(* Logix 5000 project; controller cal1632 1756-L62 rev 16.20; software revision 16.05; part 49 of 57 *)
(* tags used below, declared in another part *)
   FAULT : BOOL;
   HMI : BOOL;
   p01_recipe_active : recipe;
   p01r09_pb_global_reset : BOOL;
   p01r09_request_line_jog : BOOL;
   p01r12_master_ramped_speed : REAL;
   p01r13_line_running : BOOL;
   p01r13_line_slow_ramp : BOOL;
   p01r13_permissive_drives : BOOL;
   p02_dint_from_hmi : hmi_dint;
   p25r11_request_thread_fwd : BOOL;
   p25r11_request_thread_rev : BOOL;
   p28_ai_slitter_amps : REAL;
   p28_ai_slitter_hz : REAL;
   p28_ai_slitter_speed : REAL;
   p28_ao_sltr_selected_speed : REAL;
   p28_di_brake : BOOL;
   p28_di_motor : BOOL;
   p28_di_slitter : acs800_di_normal;
   p28_dint_to_hmi : DINT[16];
   p28_do_sltr : acs800_do_normal;
   p28_real_to_hmi : REAL[112];
   p28_slitter_on : SYS_Toggle;
   p28r06 : routine;
   p28r06_timer_fault : TIMER[4];
   p28r06_timer_warning : TIMER[4];
   p28r07 : routine;
   p28r07_timer_fault : TIMER[4];
   p28r07_timer_warning : TIMER[4];
   p28r08 : routine;
   p28r08_timer_fault : TIMER[4];
   p28r08_timer_warning : TIMER[4];
   p28r09 : routine;
   p28r09_timer_fault : TIMER[4];
   p28r09_timer_warning : TIMER[4];
   p28r11 : routine;
   p28r11_permissive_run : BOOL;
   p28r11_request_line_jog : BOOL;
   p28r11_request_run : BOOL;
   p28r11_request_thread_fwd : BOOL;
   p28r11_request_thread_rev : BOOL;
   p28r11_slitter_on : BOOL;
   p28r11_timer_fault : TIMER[10];
   p28r11_timer_warning : TIMER[5];
(* P28_Slitter, continued *)

ROUTINE R06_Real_to_HMI   (* ladder *)
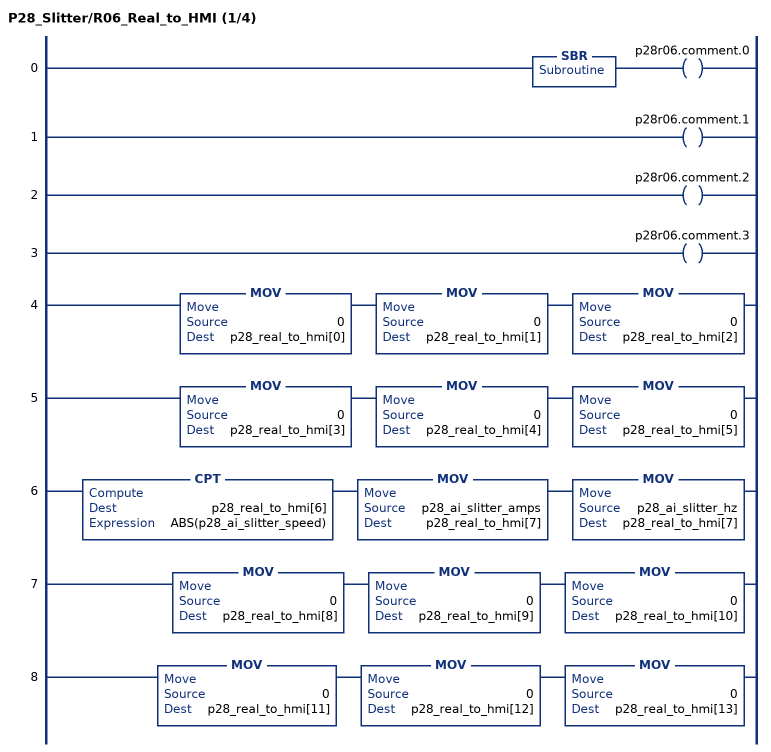
   0: SBR()OTE(p28r06.comment.0);
   1: OTE(p28r06.comment.1);
   2: OTE(p28r06.comment.2);
   3: OTE(p28r06.comment.3);
   4: MOV(0,p28_real_to_hmi[0])MOV(0,p28_real_to_hmi[1])MOV(0,p28_real_to_hmi[2]);
   5: MOV(0,p28_real_to_hmi[3])MOV(0,p28_real_to_hmi[4])MOV(0,p28_real_to_hmi[5]);
   6: CPT(p28_real_to_hmi[6],ABS(p28_ai_slitter_speed))MOV(p28_ai_slitter_amps,p28_real_to_hmi[7])MOV(p28_ai_slitter_hz,p28_real_to_hmi[7]);
   7: MOV(0,p28_real_to_hmi[8])MOV(0,p28_real_to_hmi[9])MOV(0,p28_real_to_hmi[10]);
   8: MOV(0,p28_real_to_hmi[11])MOV(0,p28_real_to_hmi[12])MOV(0,p28_real_to_hmi[13]);
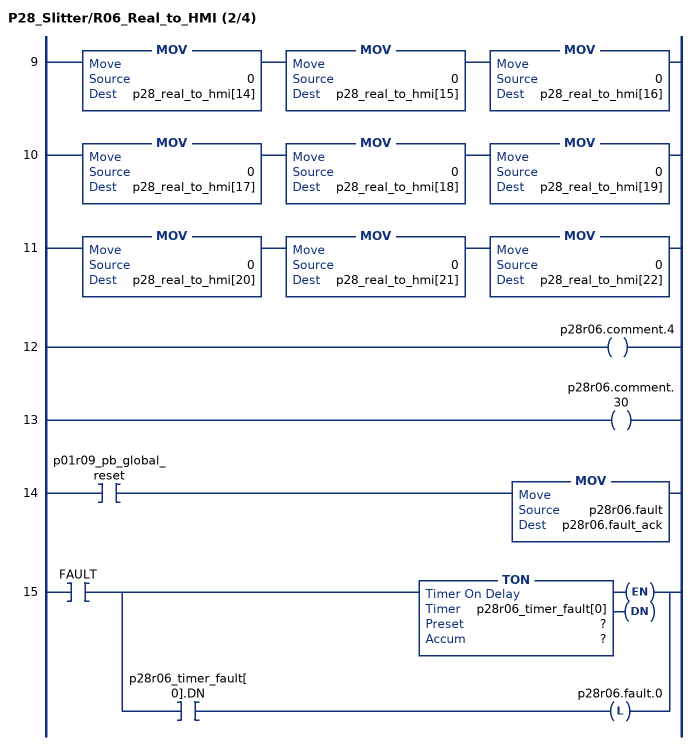
   9: MOV(0,p28_real_to_hmi[14])MOV(0,p28_real_to_hmi[15])MOV(0,p28_real_to_hmi[16]);
   10: MOV(0,p28_real_to_hmi[17])MOV(0,p28_real_to_hmi[18])MOV(0,p28_real_to_hmi[19]);
   11: MOV(0,p28_real_to_hmi[20])MOV(0,p28_real_to_hmi[21])MOV(0,p28_real_to_hmi[22]);
   12: OTE(p28r06.comment.4);
   13: OTE(p28r06.comment.30);
   14: XIC(p01r09_pb_global_reset)MOV(p28r06.fault,p28r06.fault_ack);
   15: XIC(FAULT)[TON(p28r06_timer_fault[0],?,?) ,XIC(p28r06_timer_fault[0].DN) OTL(p28r06.fault.0) ];
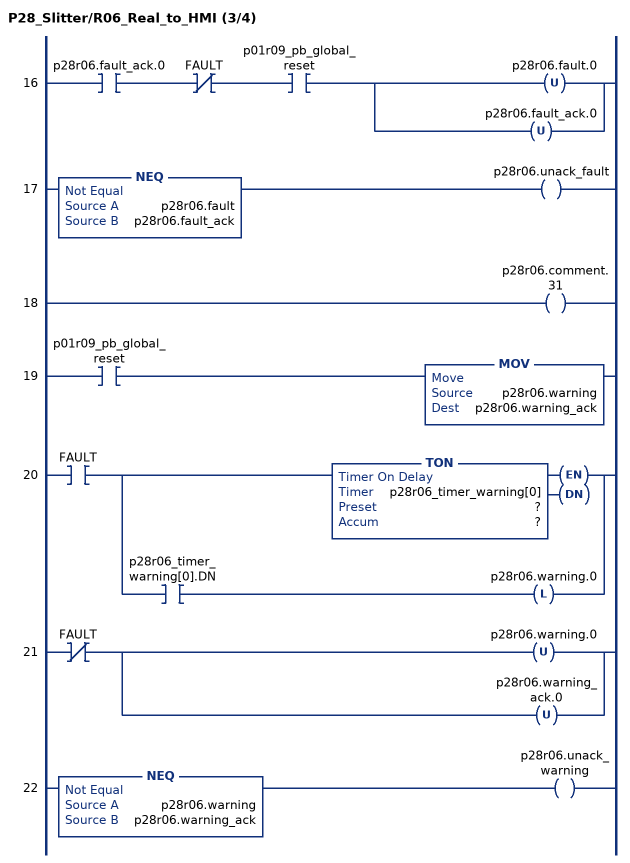
   16: XIC(p28r06.fault_ack.0)XIO(FAULT)XIC(p01r09_pb_global_reset)[OTU(p28r06.fault.0) ,OTU(p28r06.fault_ack.0) ];
   17: NEQ(p28r06.fault,p28r06.fault_ack)OTE(p28r06.unack_fault);
   18: OTE(p28r06.comment.31);
   19: XIC(p01r09_pb_global_reset)MOV(p28r06.warning,p28r06.warning_ack);
   20: XIC(FAULT)[TON(p28r06_timer_warning[0],?,?) ,XIC(p28r06_timer_warning[0].DN) OTL(p28r06.warning.0) ];
   21: XIO(FAULT)[OTU(p28r06.warning.0) ,OTU(p28r06.warning_ack.0) ];
   22: NEQ(p28r06.warning,p28r06.warning_ack)OTE(p28r06.unack_warning);
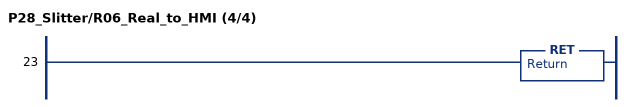
   23: RET();
END_ROUTINE

ROUTINE R07_Alarms   (* ladder *)
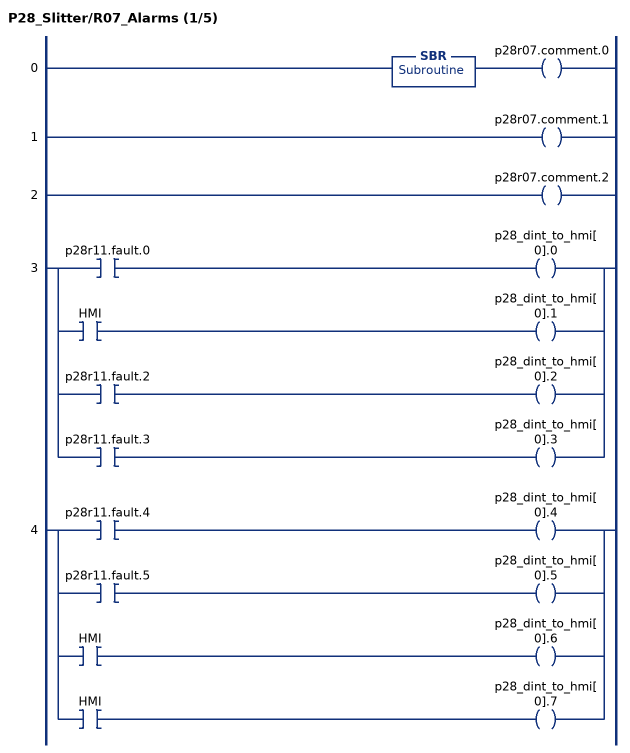
   0: SBR()OTE(p28r07.comment.0);
   1: OTE(p28r07.comment.1);
   2: OTE(p28r07.comment.2);
   3: [XIC(p28r11.fault.0) OTE(p28_dint_to_hmi[0].0) ,XIC(HMI) OTE(p28_dint_to_hmi[0].1) ,XIC(p28r11.fault.2) OTE(p28_dint_to_hmi[0].2) ,XIC(p28r11.fault.3) OTE(p28_dint_to_hmi[0].3) ];
   4: [XIC(p28r11.fault.4) OTE(p28_dint_to_hmi[0].4) ,XIC(p28r11.fault.5) OTE(p28_dint_to_hmi[0].5) ,XIC(HMI) OTE(p28_dint_to_hmi[0].6) ,XIC(HMI) OTE(p28_dint_to_hmi[0].7) ];
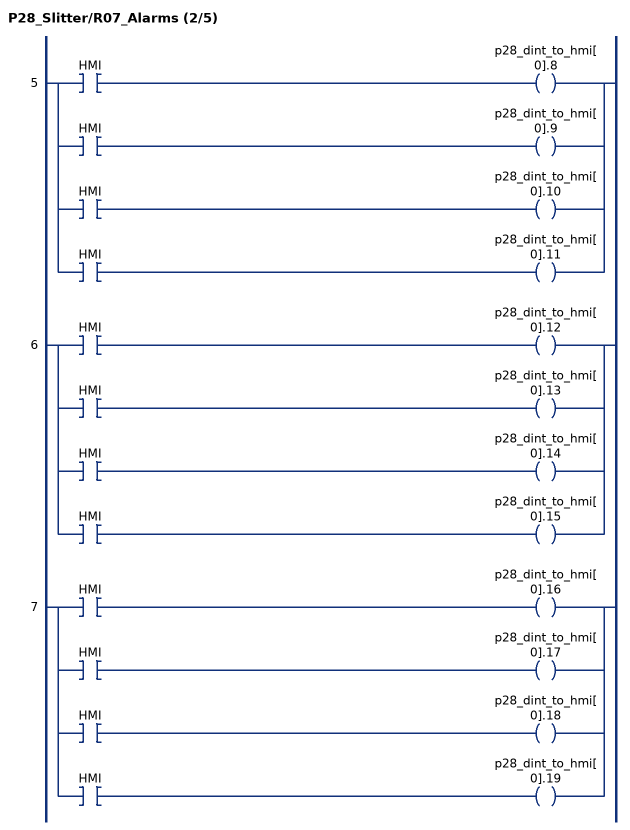
   5: [XIC(HMI) OTE(p28_dint_to_hmi[0].8) ,XIC(HMI) OTE(p28_dint_to_hmi[0].9) ,XIC(HMI) OTE(p28_dint_to_hmi[0].10) ,XIC(HMI) OTE(p28_dint_to_hmi[0].11) ];
   6: [XIC(HMI) OTE(p28_dint_to_hmi[0].12) ,XIC(HMI) OTE(p28_dint_to_hmi[0].13) ,XIC(HMI) OTE(p28_dint_to_hmi[0].14) ,XIC(HMI) OTE(p28_dint_to_hmi[0].15) ];
   7: [XIC(HMI) OTE(p28_dint_to_hmi[0].16) ,XIC(HMI) OTE(p28_dint_to_hmi[0].17) ,XIC(HMI) OTE(p28_dint_to_hmi[0].18) ,XIC(HMI) OTE(p28_dint_to_hmi[0].19) ];
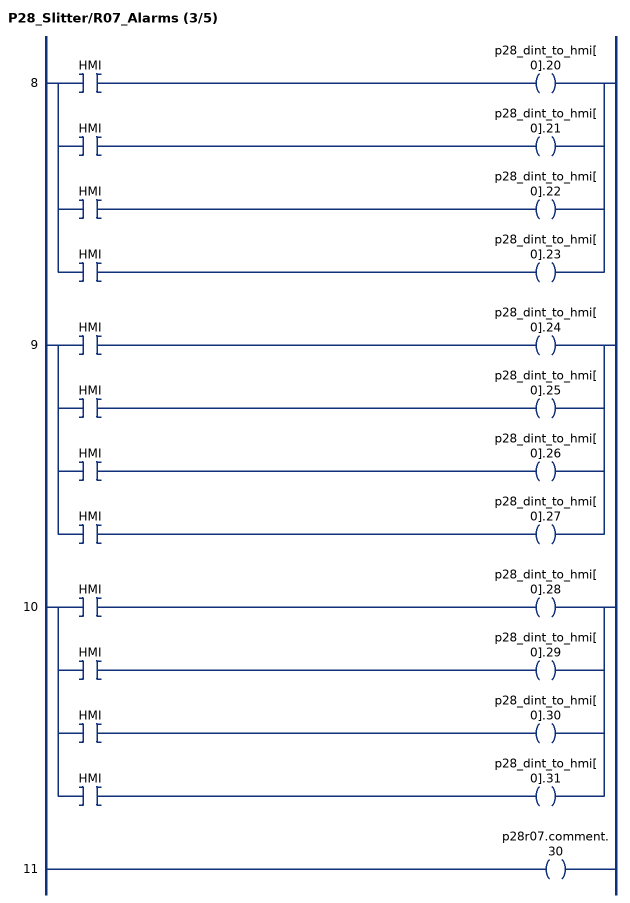
   8: [XIC(HMI) OTE(p28_dint_to_hmi[0].20) ,XIC(HMI) OTE(p28_dint_to_hmi[0].21) ,XIC(HMI) OTE(p28_dint_to_hmi[0].22) ,XIC(HMI) OTE(p28_dint_to_hmi[0].23) ];
   9: [XIC(HMI) OTE(p28_dint_to_hmi[0].24) ,XIC(HMI) OTE(p28_dint_to_hmi[0].25) ,XIC(HMI) OTE(p28_dint_to_hmi[0].26) ,XIC(HMI) OTE(p28_dint_to_hmi[0].27) ];
   10: [XIC(HMI) OTE(p28_dint_to_hmi[0].28) ,XIC(HMI) OTE(p28_dint_to_hmi[0].29) ,XIC(HMI) OTE(p28_dint_to_hmi[0].30) ,XIC(HMI) OTE(p28_dint_to_hmi[0].31) ];
   11: OTE(p28r07.comment.30);
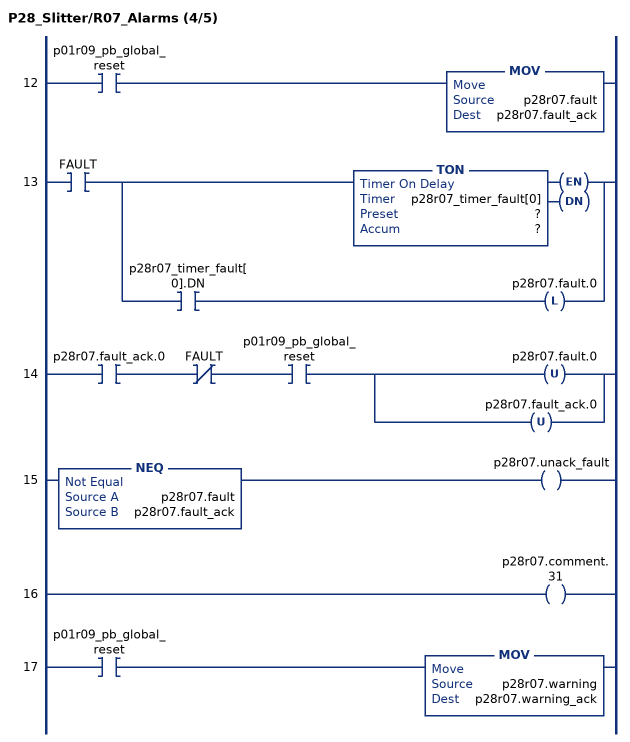
   12: XIC(p01r09_pb_global_reset)MOV(p28r07.fault,p28r07.fault_ack);
   13: XIC(FAULT)[TON(p28r07_timer_fault[0],?,?) ,XIC(p28r07_timer_fault[0].DN) OTL(p28r07.fault.0) ];
   14: XIC(p28r07.fault_ack.0)XIO(FAULT)XIC(p01r09_pb_global_reset)[OTU(p28r07.fault.0) ,OTU(p28r07.fault_ack.0) ];
   15: NEQ(p28r07.fault,p28r07.fault_ack)OTE(p28r07.unack_fault);
   16: OTE(p28r07.comment.31);
   17: XIC(p01r09_pb_global_reset)MOV(p28r07.warning,p28r07.warning_ack);
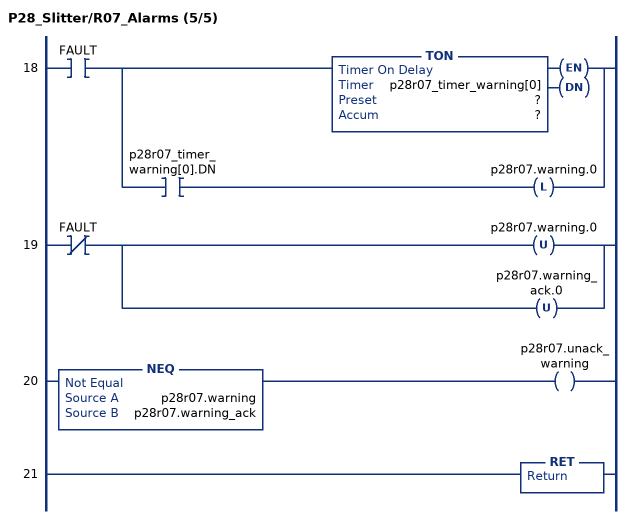
   18: XIC(FAULT)[TON(p28r07_timer_warning[0],?,?) ,XIC(p28r07_timer_warning[0].DN) OTL(p28r07.warning.0) ];
   19: XIO(FAULT)[OTU(p28r07.warning.0) ,OTU(p28r07.warning_ack.0) ];
   20: NEQ(p28r07.warning,p28r07.warning_ack)OTE(p28r07.unack_warning);
   21: RET();
END_ROUTINE

ROUTINE R08_Warnings   (* ladder *)
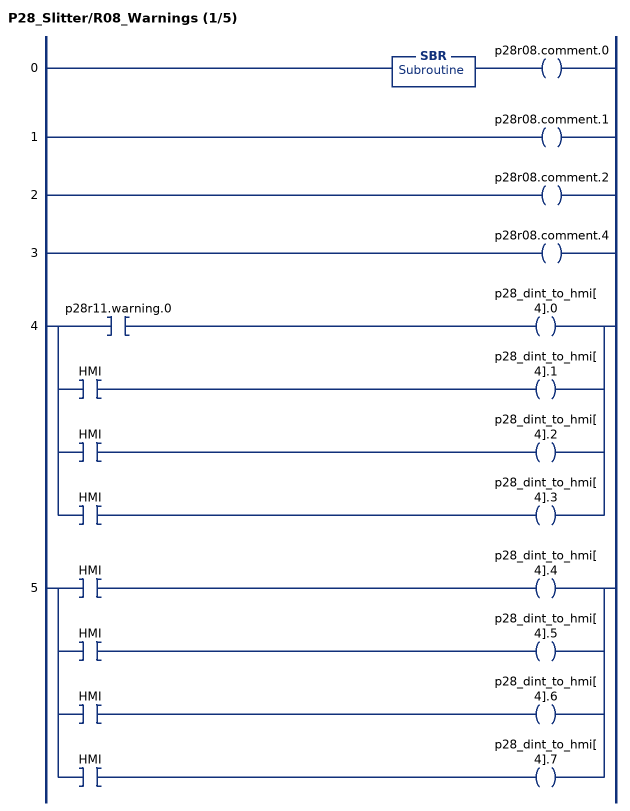
   0: SBR()OTE(p28r08.comment.0);
   1: OTE(p28r08.comment.1);
   2: OTE(p28r08.comment.2);
   3: OTE(p28r08.comment.4);
   4: [XIC(p28r11.warning.0) OTE(p28_dint_to_hmi[4].0) ,XIC(HMI) OTE(p28_dint_to_hmi[4].1) ,XIC(HMI) OTE(p28_dint_to_hmi[4].2) ,XIC(HMI) OTE(p28_dint_to_hmi[4].3) ];
   5: [XIC(HMI) OTE(p28_dint_to_hmi[4].4) ,XIC(HMI) OTE(p28_dint_to_hmi[4].5) ,XIC(HMI) OTE(p28_dint_to_hmi[4].6) ,XIC(HMI) OTE(p28_dint_to_hmi[4].7) ];
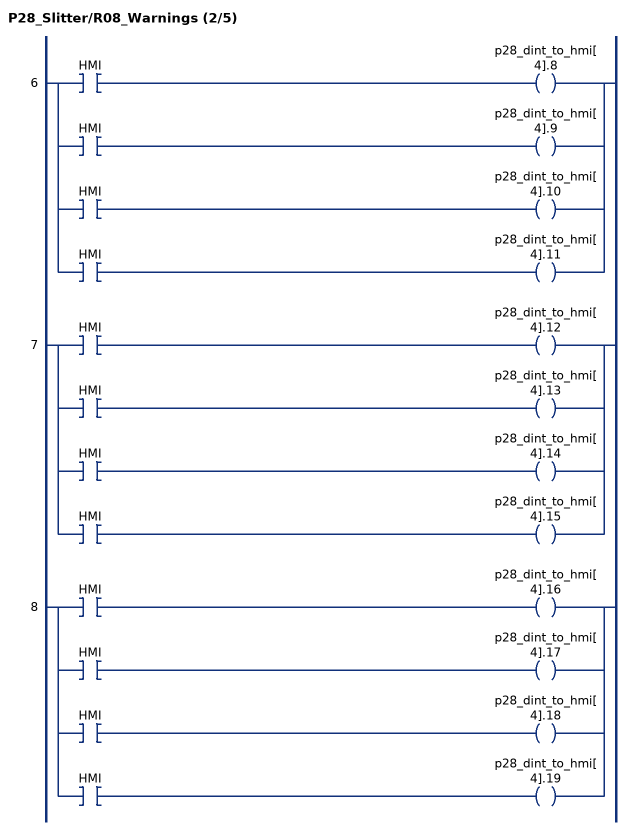
   6: [XIC(HMI) OTE(p28_dint_to_hmi[4].8) ,XIC(HMI) OTE(p28_dint_to_hmi[4].9) ,XIC(HMI) OTE(p28_dint_to_hmi[4].10) ,XIC(HMI) OTE(p28_dint_to_hmi[4].11) ];
   7: [XIC(HMI) OTE(p28_dint_to_hmi[4].12) ,XIC(HMI) OTE(p28_dint_to_hmi[4].13) ,XIC(HMI) OTE(p28_dint_to_hmi[4].14) ,XIC(HMI) OTE(p28_dint_to_hmi[4].15) ];
   8: [XIC(HMI) OTE(p28_dint_to_hmi[4].16) ,XIC(HMI) OTE(p28_dint_to_hmi[4].17) ,XIC(HMI) OTE(p28_dint_to_hmi[4].18) ,XIC(HMI) OTE(p28_dint_to_hmi[4].19) ];
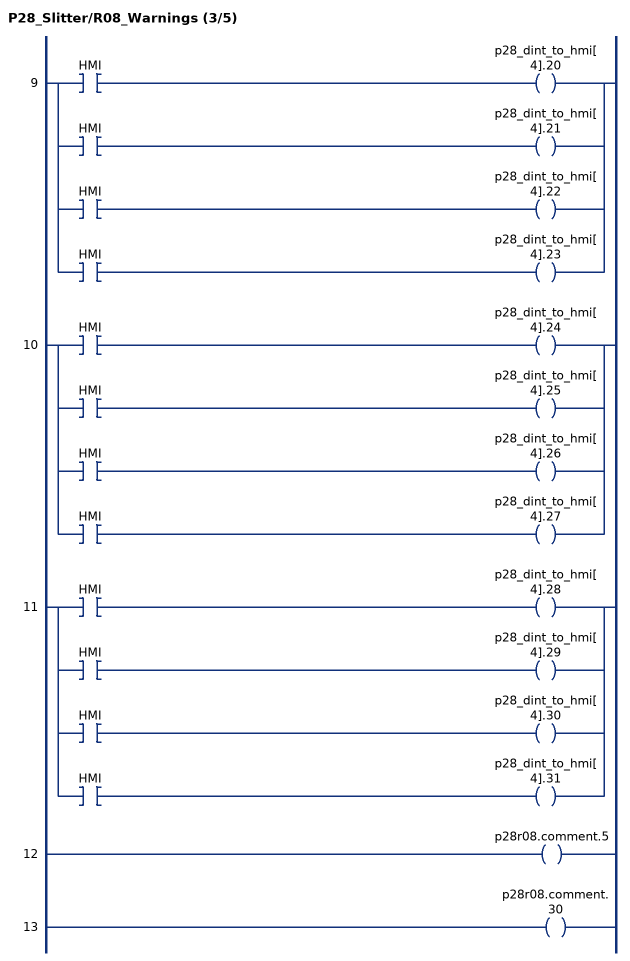
   9: [XIC(HMI) OTE(p28_dint_to_hmi[4].20) ,XIC(HMI) OTE(p28_dint_to_hmi[4].21) ,XIC(HMI) OTE(p28_dint_to_hmi[4].22) ,XIC(HMI) OTE(p28_dint_to_hmi[4].23) ];
   10: [XIC(HMI) OTE(p28_dint_to_hmi[4].24) ,XIC(HMI) OTE(p28_dint_to_hmi[4].25) ,XIC(HMI) OTE(p28_dint_to_hmi[4].26) ,XIC(HMI) OTE(p28_dint_to_hmi[4].27) ];
   11: [XIC(HMI) OTE(p28_dint_to_hmi[4].28) ,XIC(HMI) OTE(p28_dint_to_hmi[4].29) ,XIC(HMI) OTE(p28_dint_to_hmi[4].30) ,XIC(HMI) OTE(p28_dint_to_hmi[4].31) ];
   12: OTE(p28r08.comment.5);
   13: OTE(p28r08.comment.30);
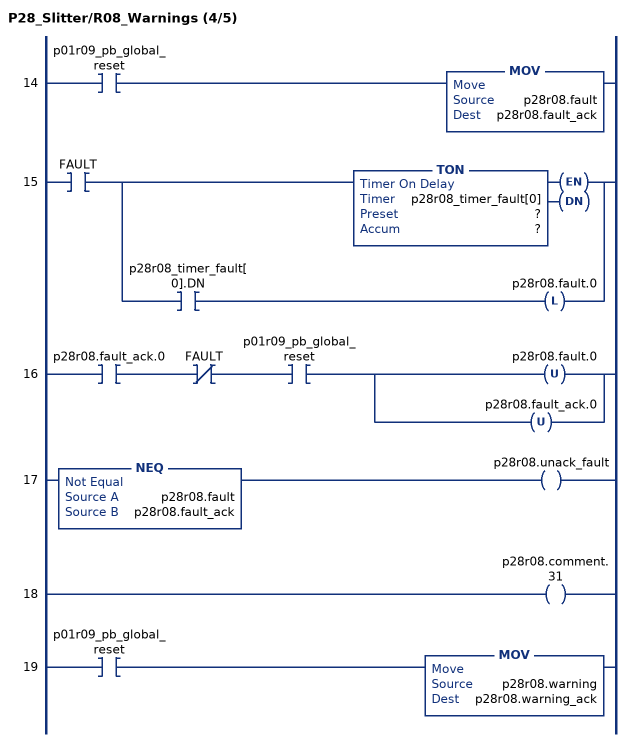
   14: XIC(p01r09_pb_global_reset)MOV(p28r08.fault,p28r08.fault_ack);
   15: XIC(FAULT)[TON(p28r08_timer_fault[0],?,?) ,XIC(p28r08_timer_fault[0].DN) OTL(p28r08.fault.0) ];
   16: XIC(p28r08.fault_ack.0)XIO(FAULT)XIC(p01r09_pb_global_reset)[OTU(p28r08.fault.0) ,OTU(p28r08.fault_ack.0) ];
   17: NEQ(p28r08.fault,p28r08.fault_ack)OTE(p28r08.unack_fault);
   18: OTE(p28r08.comment.31);
   19: XIC(p01r09_pb_global_reset)MOV(p28r08.warning,p28r08.warning_ack);
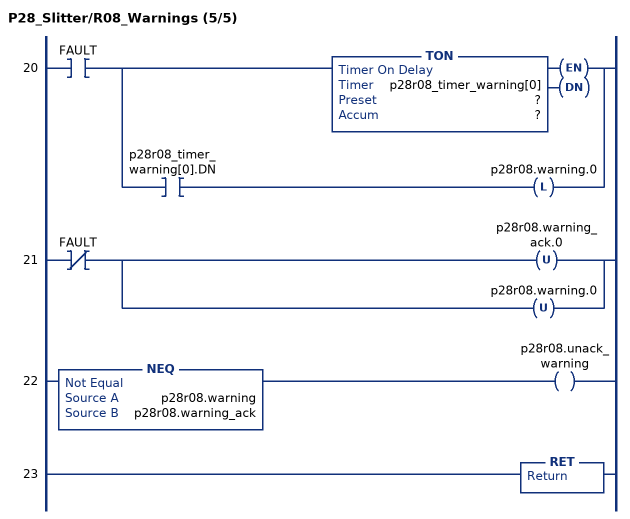
   20: XIC(FAULT)[TON(p28r08_timer_warning[0],?,?) ,XIC(p28r08_timer_warning[0].DN) OTL(p28r08.warning.0) ];
   21: XIO(FAULT)[OTU(p28r08.warning_ack.0) ,OTU(p28r08.warning.0) ];
   22: NEQ(p28r08.warning,p28r08.warning_ack)OTE(p28r08.unack_warning);
   23: RET();
END_ROUTINE

ROUTINE R09_Modes   (* ladder *)
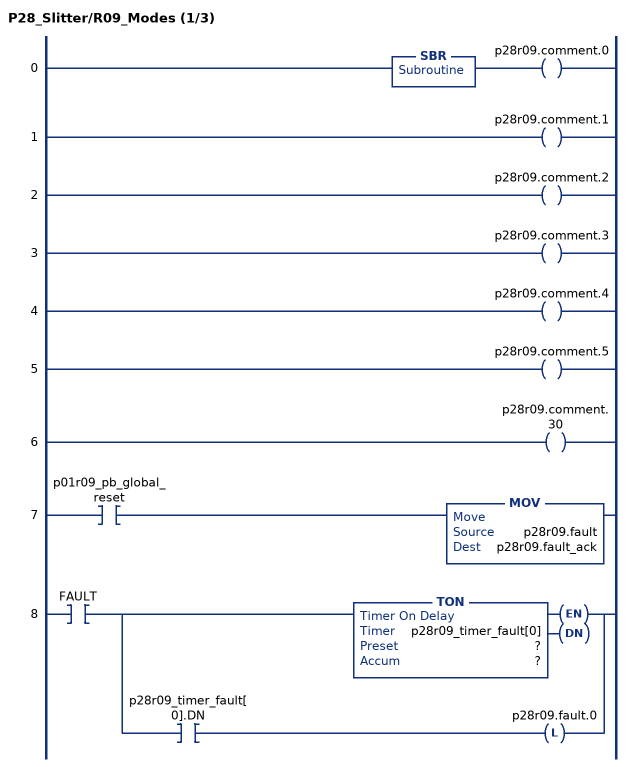
   0: SBR()OTE(p28r09.comment.0);
   1: OTE(p28r09.comment.1);
   2: OTE(p28r09.comment.2);
   3: OTE(p28r09.comment.3);
   4: OTE(p28r09.comment.4);
   5: OTE(p28r09.comment.5);
   6: OTE(p28r09.comment.30);
   7: XIC(p01r09_pb_global_reset)MOV(p28r09.fault,p28r09.fault_ack);
   8: XIC(FAULT)[TON(p28r09_timer_fault[0],?,?) ,XIC(p28r09_timer_fault[0].DN) OTL(p28r09.fault.0) ];
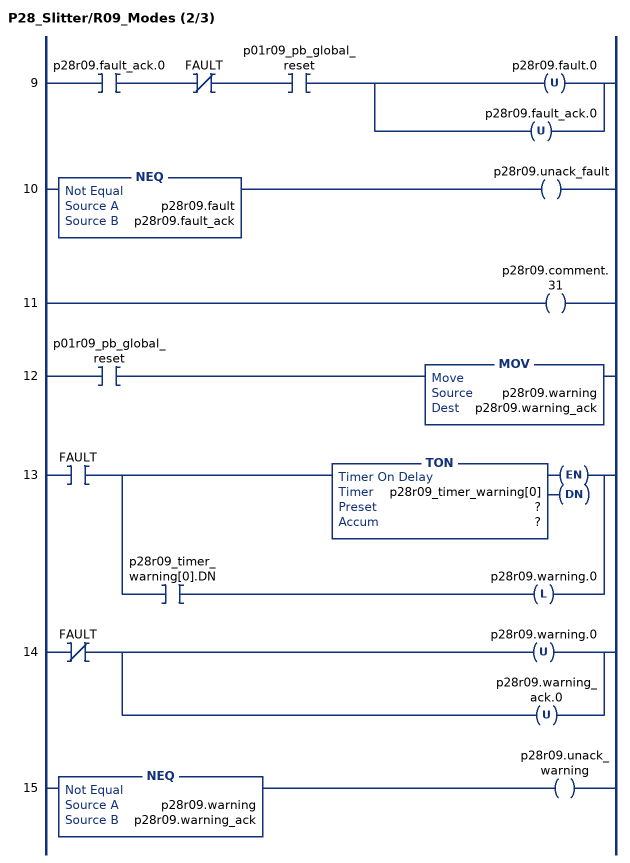
   9: XIC(p28r09.fault_ack.0)XIO(FAULT)XIC(p01r09_pb_global_reset)[OTU(p28r09.fault.0) ,OTU(p28r09.fault_ack.0) ];
   10: NEQ(p28r09.fault,p28r09.fault_ack)OTE(p28r09.unack_fault);
   11: OTE(p28r09.comment.31);
   12: XIC(p01r09_pb_global_reset)MOV(p28r09.warning,p28r09.warning_ack);
   13: XIC(FAULT)[TON(p28r09_timer_warning[0],?,?) ,XIC(p28r09_timer_warning[0].DN) OTL(p28r09.warning.0) ];
   14: XIO(FAULT)[OTU(p28r09.warning.0) ,OTU(p28r09.warning_ack.0) ];
   15: NEQ(p28r09.warning,p28r09.warning_ack)OTE(p28r09.unack_warning);
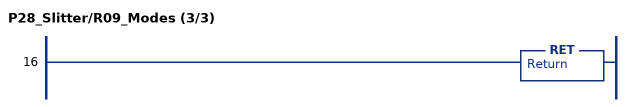
   16: RET();
END_ROUTINE

ROUTINE R11_VFD   (* ladder *)
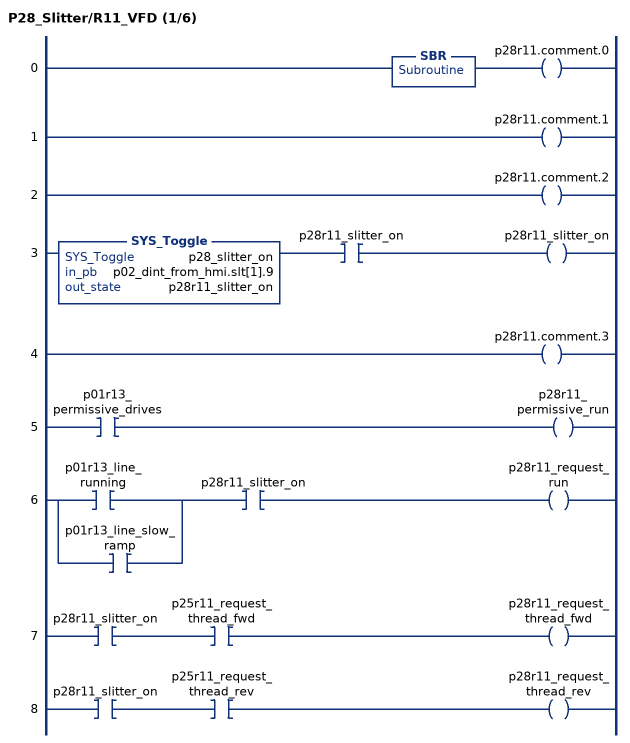
   0: SBR()OTE(p28r11.comment.0);
   1: OTE(p28r11.comment.1);
   2: OTE(p28r11.comment.2);
   3: SYS_Toggle(p28_slitter_on,p02_dint_from_hmi.slt[1].9,p28r11_slitter_on)XIC(p28r11_slitter_on)OTE(p28r11_slitter_on);
   4: OTE(p28r11.comment.3);
   5: XIC(p01r13_permissive_drives)OTE(p28r11_permissive_run);
   6: [XIC(p01r13_line_running) ,XIC(p01r13_line_slow_ramp) ]XIC(p28r11_slitter_on)OTE(p28r11_request_run);
   7: XIC(p28r11_slitter_on)XIC(p25r11_request_thread_fwd)OTE(p28r11_request_thread_fwd);
   8: XIC(p28r11_slitter_on)XIC(p25r11_request_thread_rev)OTE(p28r11_request_thread_rev);
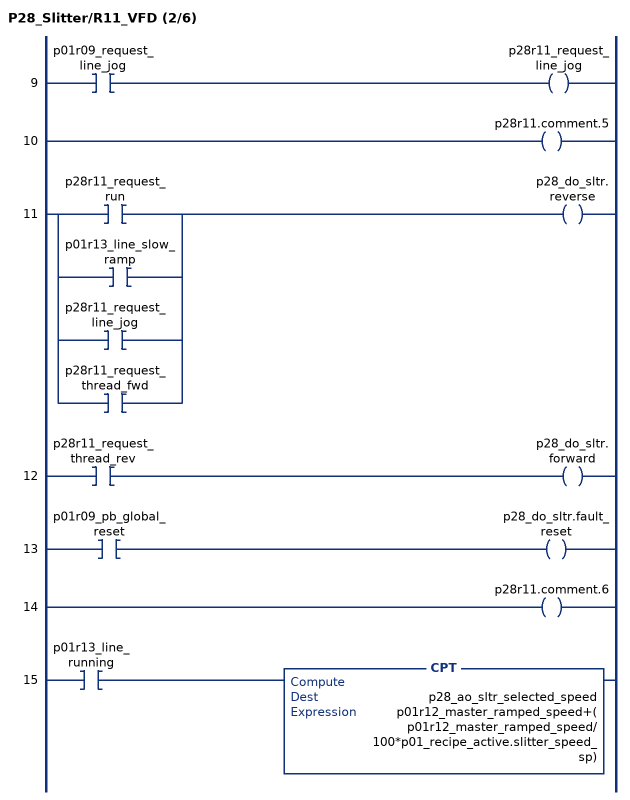
   9: XIC(p01r09_request_line_jog)OTE(p28r11_request_line_jog);
   10: OTE(p28r11.comment.5);
   11: [XIC(p28r11_request_run) ,XIC(p01r13_line_slow_ramp) ,XIC(p28r11_request_line_jog) ,XIC(p28r11_request_thread_fwd) ]OTE(p28_do_sltr.reverse);
   12: XIC(p28r11_request_thread_rev)OTE(p28_do_sltr.forward);
   13: XIC(p01r09_pb_global_reset)OTE(p28_do_sltr.fault_reset);
   14: OTE(p28r11.comment.6);
   15: XIC(p01r13_line_running)CPT(p28_ao_sltr_selected_speed,p01r12_master_ramped_speed+(p01r12_master_ramped_speed/100*p01_recipe_active.slitter_speed_sp));
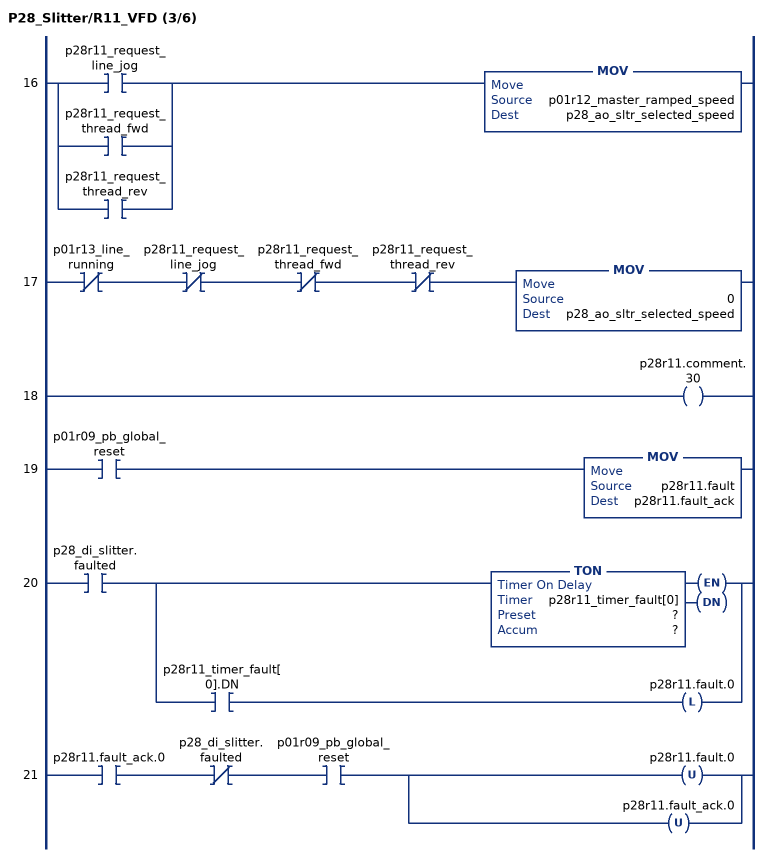
   16: [XIC(p28r11_request_line_jog) ,XIC(p28r11_request_thread_fwd) ,XIC(p28r11_request_thread_rev) ]MOV(p01r12_master_ramped_speed,p28_ao_sltr_selected_speed);
   17: XIO(p01r13_line_running)XIO(p28r11_request_line_jog)XIO(p28r11_request_thread_fwd)XIO(p28r11_request_thread_rev)MOV(0,p28_ao_sltr_selected_speed);
   18: OTE(p28r11.comment.30);
   19: XIC(p01r09_pb_global_reset)MOV(p28r11.fault,p28r11.fault_ack);
   20: XIC(p28_di_slitter.faulted)[TON(p28r11_timer_fault[0],?,?) ,XIC(p28r11_timer_fault[0].DN) OTL(p28r11.fault.0) ];
   21: XIC(p28r11.fault_ack.0)XIO(p28_di_slitter.faulted)XIC(p01r09_pb_global_reset)[OTU(p28r11.fault.0) ,OTU(p28r11.fault_ack.0) ];
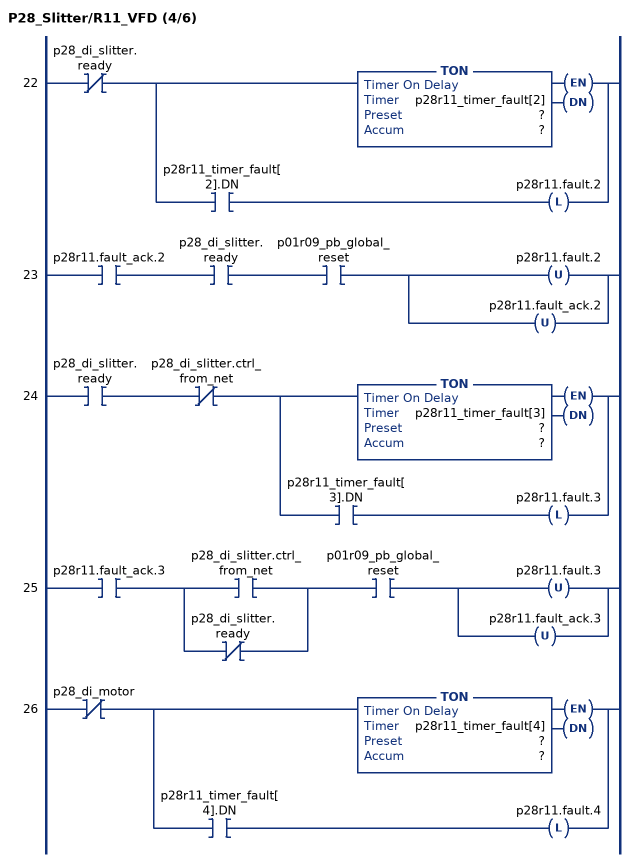
   22: XIO(p28_di_slitter.ready)[TON(p28r11_timer_fault[2],?,?) ,XIC(p28r11_timer_fault[2].DN) OTL(p28r11.fault.2) ];
   23: XIC(p28r11.fault_ack.2)XIC(p28_di_slitter.ready)XIC(p01r09_pb_global_reset)[OTU(p28r11.fault.2) ,OTU(p28r11.fault_ack.2) ];
   24: XIC(p28_di_slitter.ready)XIO(p28_di_slitter.ctrl_from_net)[TON(p28r11_timer_fault[3],?,?) ,XIC(p28r11_timer_fault[3].DN) OTL(p28r11.fault.3) ];
   25: XIC(p28r11.fault_ack.3)[XIC(p28_di_slitter.ctrl_from_net) ,XIO(p28_di_slitter.ready) ]XIC(p01r09_pb_global_reset)[OTU(p28r11.fault.3) ,OTU(p28r11.fault_ack.3) ];
   26: XIO(p28_di_motor)[TON(p28r11_timer_fault[4],?,?) ,XIC(p28r11_timer_fault[4].DN) OTL(p28r11.fault.4) ];
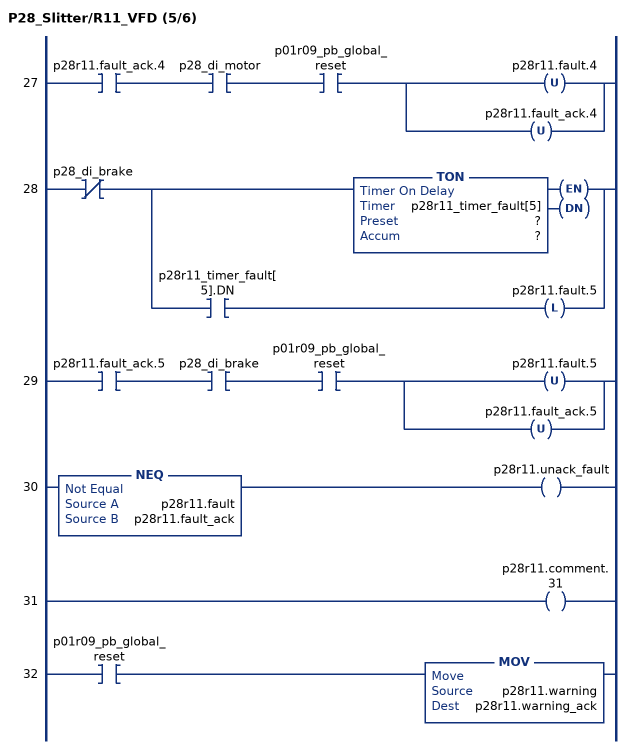
   27: XIC(p28r11.fault_ack.4)XIC(p28_di_motor)XIC(p01r09_pb_global_reset)[OTU(p28r11.fault.4) ,OTU(p28r11.fault_ack.4) ];
   28: XIO(p28_di_brake)[TON(p28r11_timer_fault[5],?,?) ,XIC(p28r11_timer_fault[5].DN) OTL(p28r11.fault.5) ];
   29: XIC(p28r11.fault_ack.5)XIC(p28_di_brake)XIC(p01r09_pb_global_reset)[OTU(p28r11.fault.5) ,OTU(p28r11.fault_ack.5) ];
   30: NEQ(p28r11.fault,p28r11.fault_ack)OTE(p28r11.unack_fault);
   31: OTE(p28r11.comment.31);
   32: XIC(p01r09_pb_global_reset)MOV(p28r11.warning,p28r11.warning_ack);
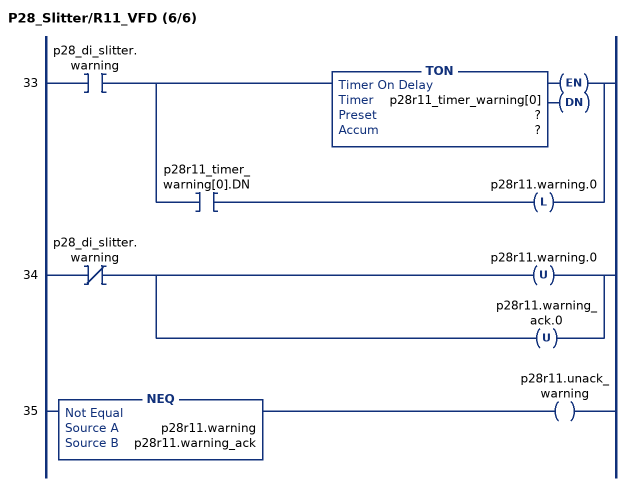
   33: XIC(p28_di_slitter.warning)[TON(p28r11_timer_warning[0],?,?) ,XIC(p28r11_timer_warning[0].DN) OTL(p28r11.warning.0) ];
   34: XIO(p28_di_slitter.warning)[OTU(p28r11.warning.0) ,OTU(p28r11.warning_ack.0) ];
   35: NEQ(p28r11.warning,p28r11.warning_ack)OTE(p28r11.unack_warning);
END_ROUTINE
END_PROGRAM
